// TIA Portal V16 export
// export: Created 2023-01-31T04:00:58.1302964Z, ExportSetting WithDefaults, WithReadOnly, DisplayName Totally Integrated Automation Portal, DisplayVersion V16 Update 1, DisplayName TIA Portal Version Control Interface, DisplayVersion V16, DisplayName TIA Portal Openness, DisplayVersion V16 Update 1, DisplayName SINAMICS Startdrive Advanced, DisplayVersion V16, DisplayName SINAMICS Startdrive G130, G150, S120, S150, SINAMICS MV, S210, DisplayVersion V16, DisplayName SINAMICS Startdrive G110M, G120, G120C, G120D, G120P, DisplayVersion V16, DisplayName STEP 7 Professional, DisplayVersion V16 Update 1, DisplayName STEP 7 Safety, DisplayVersion V16, DisplayName WinCC Advanced, DisplayVersion V16 Update 1
FUNCTION "022SAE001_Call" : Void   // FC80, LAD
TITLE = 022SAE001 Deposit 1 / 010ABS001 Ablage 1
{ S7_Optimized_Access := 'FALSE' }
VERSION : 0.1
// stored: AutoNumber true, CodeModifiedDate 2021-01-26T01:38:20.3874578Z, CompileDate 2021-02-05T02:55:14.1436684Z, CreationDate 2019-06-27T08:21:26.7500417Z, HandleErrorsWithinBlock false, InterfaceModifiedDate 2017-10-27T11:23:23.7919428Z, IsConsistent true, IsIECCheckEnabled false, IsKnowHowProtected false, IsWriteProtected false, LibraryConformanceStatus Error: The block contains calls of single instances. Warning: The object contains access to global data blocks. Warning: The block contains direct access to inputs, outputs, bit memories, indirect access to the registry or indirect access to external memory areas that are unknown at the time of compilation., ModifiedDate 2021-01-26T01:38:20.3874578Z, ParameterModified 2017-10-27T11:23:23.7469402Z, PLCSimAdvancedSupport true, SetENOAutomatically false, StructureModified 2017-10-27T11:23:23.7919428Z, UDAEnableTagReadback false
   VAR_TEMP   // added for the SCL form of the ladder/FBD networks
      _w1 : Bool;
      _s5time1 : S5Time;
   END_VAR
BEGIN

REGION Network 1: 022SAE001-BZ1.1 part control
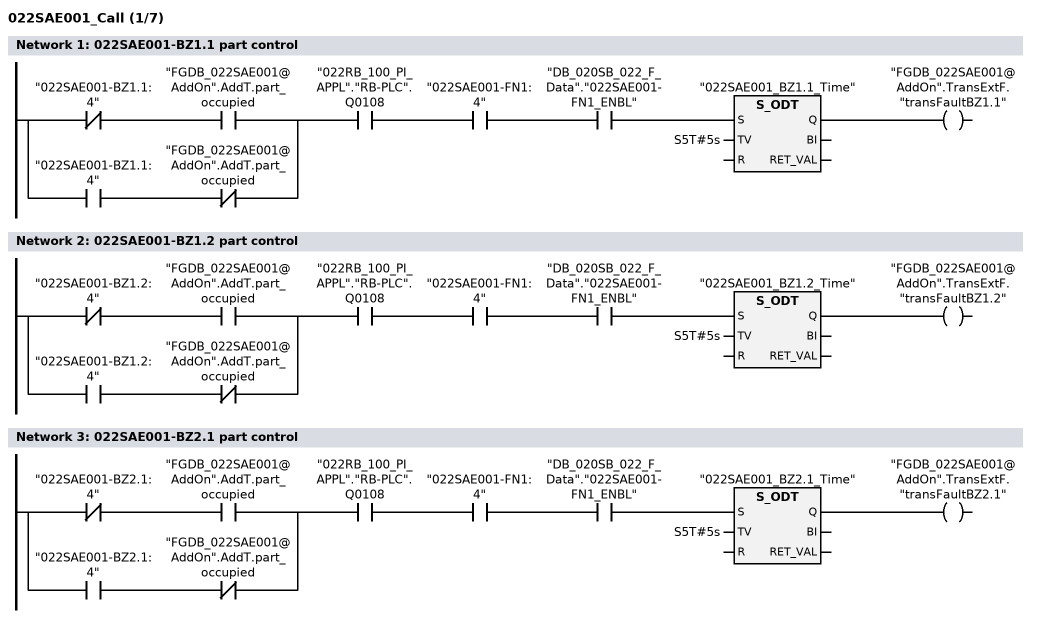
   RUNG wire#powerrail
      I_Contact( "022SAE001-BZ1.1:4" )
      Contact( "FGDB_022SAE001@AddOn".AddT.part_occupied )
      wire#w1
      Contact( "022RB_100_PI_APPL"."RB-PLC".Q0108 )
      Contact( "022SAE001-FN1:4" )
      Contact( "DB_020SB_022_F_Data"."022SAE001-FN1_ENBL" )
      S_ODT(T_NO := "022SAE001_BZ1.1_Time", TV := S5T#5s, R :=, BI =>, RET_VAL =>)
      Coil( "FGDB_022SAE001@AddOn".TransExtF."transFaultBZ1.1" )
   END_RUNG
   RUNG wire#powerrail
      Contact( "022SAE001-BZ1.1:4" )
      I_Contact( "FGDB_022SAE001@AddOn".AddT.part_occupied )
   END_RUNG wire#w1
   // the same network as SCL:
   #_s5time1 := S_ODT(T_NO := "022SAE001_BZ1.1_Time",
                      S := ((NOT "022SAE001-BZ1.1:4" AND "FGDB_022SAE001@AddOn".AddT.part_occupied) OR ("022SAE001-BZ1.1:4" AND NOT "FGDB_022SAE001@AddOn".AddT.part_occupied)) AND "022RB_100_PI_APPL"."RB-PLC".Q0108 AND "022SAE001-FN1:4" AND "DB_020SB_022_F_Data"."022SAE001-FN1_ENBL",
                      TV := S5T#5s,
                      Q => #_w1);
   "FGDB_022SAE001@AddOn".TransExtF."transFaultBZ1.1" := #_w1;
END_REGION

REGION Network 2: 022SAE001-BZ1.2 part control
   RUNG wire#powerrail
      I_Contact( "022SAE001-BZ1.2:4" )
      Contact( "FGDB_022SAE001@AddOn".AddT.part_occupied )
      wire#w1
      Contact( "022RB_100_PI_APPL"."RB-PLC".Q0108 )
      Contact( "022SAE001-FN1:4" )
      Contact( "DB_020SB_022_F_Data"."022SAE001-FN1_ENBL" )
      S_ODT(T_NO := "022SAE001_BZ1.2_Time", TV := S5T#5s, R :=, BI =>, RET_VAL =>)
      Coil( "FGDB_022SAE001@AddOn".TransExtF."transFaultBZ1.2" )
   END_RUNG
   RUNG wire#powerrail
      Contact( "022SAE001-BZ1.2:4" )
      I_Contact( "FGDB_022SAE001@AddOn".AddT.part_occupied )
   END_RUNG wire#w1
   // the same network as SCL:
   #_s5time1 := S_ODT(T_NO := "022SAE001_BZ1.2_Time",
                      S := ((NOT "022SAE001-BZ1.2:4" AND "FGDB_022SAE001@AddOn".AddT.part_occupied) OR ("022SAE001-BZ1.2:4" AND NOT "FGDB_022SAE001@AddOn".AddT.part_occupied)) AND "022RB_100_PI_APPL"."RB-PLC".Q0108 AND "022SAE001-FN1:4" AND "DB_020SB_022_F_Data"."022SAE001-FN1_ENBL",
                      TV := S5T#5s,
                      Q => #_w1);
   "FGDB_022SAE001@AddOn".TransExtF."transFaultBZ1.2" := #_w1;
END_REGION

REGION Network 3: 022SAE001-BZ2.1 part control
   RUNG wire#powerrail
      I_Contact( "022SAE001-BZ2.1:4" )
      Contact( "FGDB_022SAE001@AddOn".AddT.part_occupied )
      wire#w1
      Contact( "022RB_100_PI_APPL"."RB-PLC".Q0108 )
      Contact( "022SAE001-FN1:4" )
      Contact( "DB_020SB_022_F_Data"."022SAE001-FN1_ENBL" )
      S_ODT(T_NO := "022SAE001_BZ2.1_Time", TV := S5T#5s, R :=, BI =>, RET_VAL =>)
      Coil( "FGDB_022SAE001@AddOn".TransExtF."transFaultBZ2.1" )
   END_RUNG
   RUNG wire#powerrail
      Contact( "022SAE001-BZ2.1:4" )
      I_Contact( "FGDB_022SAE001@AddOn".AddT.part_occupied )
   END_RUNG wire#w1
   // the same network as SCL:
   #_s5time1 := S_ODT(T_NO := "022SAE001_BZ2.1_Time",
                      S := ((NOT "022SAE001-BZ2.1:4" AND "FGDB_022SAE001@AddOn".AddT.part_occupied) OR ("022SAE001-BZ2.1:4" AND NOT "FGDB_022SAE001@AddOn".AddT.part_occupied)) AND "022RB_100_PI_APPL"."RB-PLC".Q0108 AND "022SAE001-FN1:4" AND "DB_020SB_022_F_Data"."022SAE001-FN1_ENBL",
                      TV := S5T#5s,
                      Q => #_w1);
   "FGDB_022SAE001@AddOn".TransExtF."transFaultBZ2.1" := #_w1;
END_REGION

REGION Network 4: Enter additional malfunctions 022SAE001
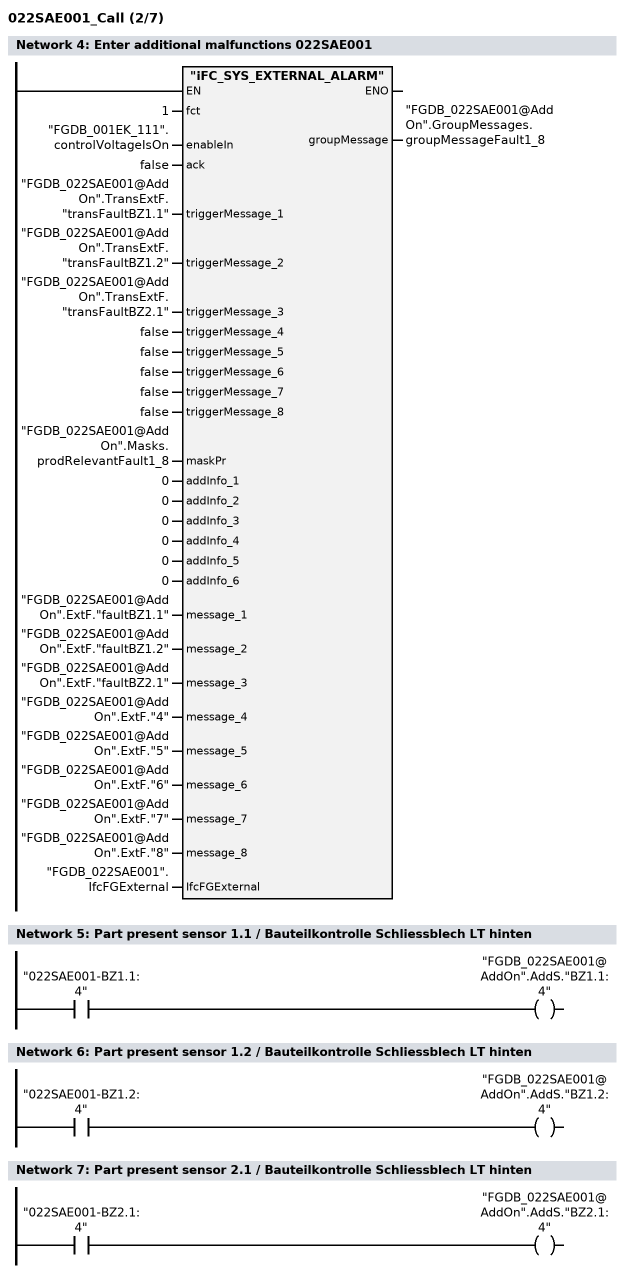
   RUNG wire#powerrail
      "iFC_SYS_EXTERNAL_ALARM"(fct := 1, enableIn := "FGDB_001EK_111".controlVoltageIsOn, ack := false, triggerMessage_1 := "FGDB_022SAE001@AddOn".TransExtF."transFaultBZ1.1", triggerMessage_2 := "FGDB_022SAE001@AddOn".TransExtF."transFaultBZ1.2", triggerMessage_3 := "FGDB_022SAE001@AddOn".TransExtF."transFaultBZ2.1", triggerMessage_4 := false, triggerMessage_5 := false, triggerMessage_6 := false, triggerMessage_7 := false, triggerMessage_8 := false, maskPr := "FGDB_022SAE001@AddOn".Masks.prodRelevantFault1_8, addInfo_1 := 0, addInfo_2 := 0, addInfo_3 := 0, addInfo_4 := 0, addInfo_5 := 0, addInfo_6 := 0, message_1 := "FGDB_022SAE001@AddOn".ExtF."faultBZ1.1", message_2 := "FGDB_022SAE001@AddOn".ExtF."faultBZ1.2", message_3 := "FGDB_022SAE001@AddOn".ExtF."faultBZ2.1", message_4 := "FGDB_022SAE001@AddOn".ExtF."4", message_5 := "FGDB_022SAE001@AddOn".ExtF."5", message_6 := "FGDB_022SAE001@AddOn".ExtF."6", message_7 := "FGDB_022SAE001@AddOn".ExtF."7", message_8 := "FGDB_022SAE001@AddOn".ExtF."8", IfcFGExternal := "FGDB_022SAE001".IfcFGExternal, groupMessage => "FGDB_022SAE001@AddOn".GroupMessages.groupMessageFault1_8)
   END_RUNG
   // the same network as SCL:
   "iFC_SYS_EXTERNAL_ALARM"(fct := 1,
                           enableIn := "FGDB_001EK_111".controlVoltageIsOn,
                           ack := false,
                           triggerMessage_1 := "FGDB_022SAE001@AddOn".TransExtF."transFaultBZ1.1",
                           triggerMessage_2 := "FGDB_022SAE001@AddOn".TransExtF."transFaultBZ1.2",
                           triggerMessage_3 := "FGDB_022SAE001@AddOn".TransExtF."transFaultBZ2.1",
                           triggerMessage_4 := false,
                           triggerMessage_5 := false,
                           triggerMessage_6 := false,
                           triggerMessage_7 := false,
                           triggerMessage_8 := false,
                           maskPr := "FGDB_022SAE001@AddOn".Masks.prodRelevantFault1_8,
                           addInfo_1 := 0,
                           addInfo_2 := 0,
                           addInfo_3 := 0,
                           addInfo_4 := 0,
                           addInfo_5 := 0,
                           addInfo_6 := 0,
                           message_1 := "FGDB_022SAE001@AddOn".ExtF."faultBZ1.1",
                           message_2 := "FGDB_022SAE001@AddOn".ExtF."faultBZ1.2",
                           message_3 := "FGDB_022SAE001@AddOn".ExtF."faultBZ2.1",
                           message_4 := "FGDB_022SAE001@AddOn".ExtF."4",
                           message_5 := "FGDB_022SAE001@AddOn".ExtF."5",
                           message_6 := "FGDB_022SAE001@AddOn".ExtF."6",
                           message_7 := "FGDB_022SAE001@AddOn".ExtF."7",
                           message_8 := "FGDB_022SAE001@AddOn".ExtF."8",
                           IfcFGExternal := "FGDB_022SAE001".IfcFGExternal,
                           groupMessage => "FGDB_022SAE001@AddOn".GroupMessages.groupMessageFault1_8);
END_REGION

REGION Network 5: Part present sensor 1.1 / Bauteilkontrolle Schliessblech LT hinten
   RUNG wire#powerrail
      Contact( "022SAE001-BZ1.1:4" )
      Coil( "FGDB_022SAE001@AddOn".AddS."BZ1.1:4" )
   END_RUNG
   // the same network as SCL:
   "FGDB_022SAE001@AddOn".AddS."BZ1.1:4" := "022SAE001-BZ1.1:4";
END_REGION

REGION Network 6: Part present sensor 1.2 / Bauteilkontrolle Schliessblech LT hinten
   RUNG wire#powerrail
      Contact( "022SAE001-BZ1.2:4" )
      Coil( "FGDB_022SAE001@AddOn".AddS."BZ1.2:4" )
   END_RUNG
   // the same network as SCL:
   "FGDB_022SAE001@AddOn".AddS."BZ1.2:4" := "022SAE001-BZ1.2:4";
END_REGION

REGION Network 7: Part present sensor 2.1 / Bauteilkontrolle Schliessblech LT hinten
   RUNG wire#powerrail
      Contact( "022SAE001-BZ2.1:4" )
      Coil( "FGDB_022SAE001@AddOn".AddS."BZ2.1:4" )
   END_RUNG
   // the same network as SCL:
   "FGDB_022SAE001@AddOn".AddS."BZ2.1:4" := "022SAE001-BZ2.1:4";
END_REGION

REGION Network 8: 022SAE001 Part1 occupied / Teil belegt Federbeintopf
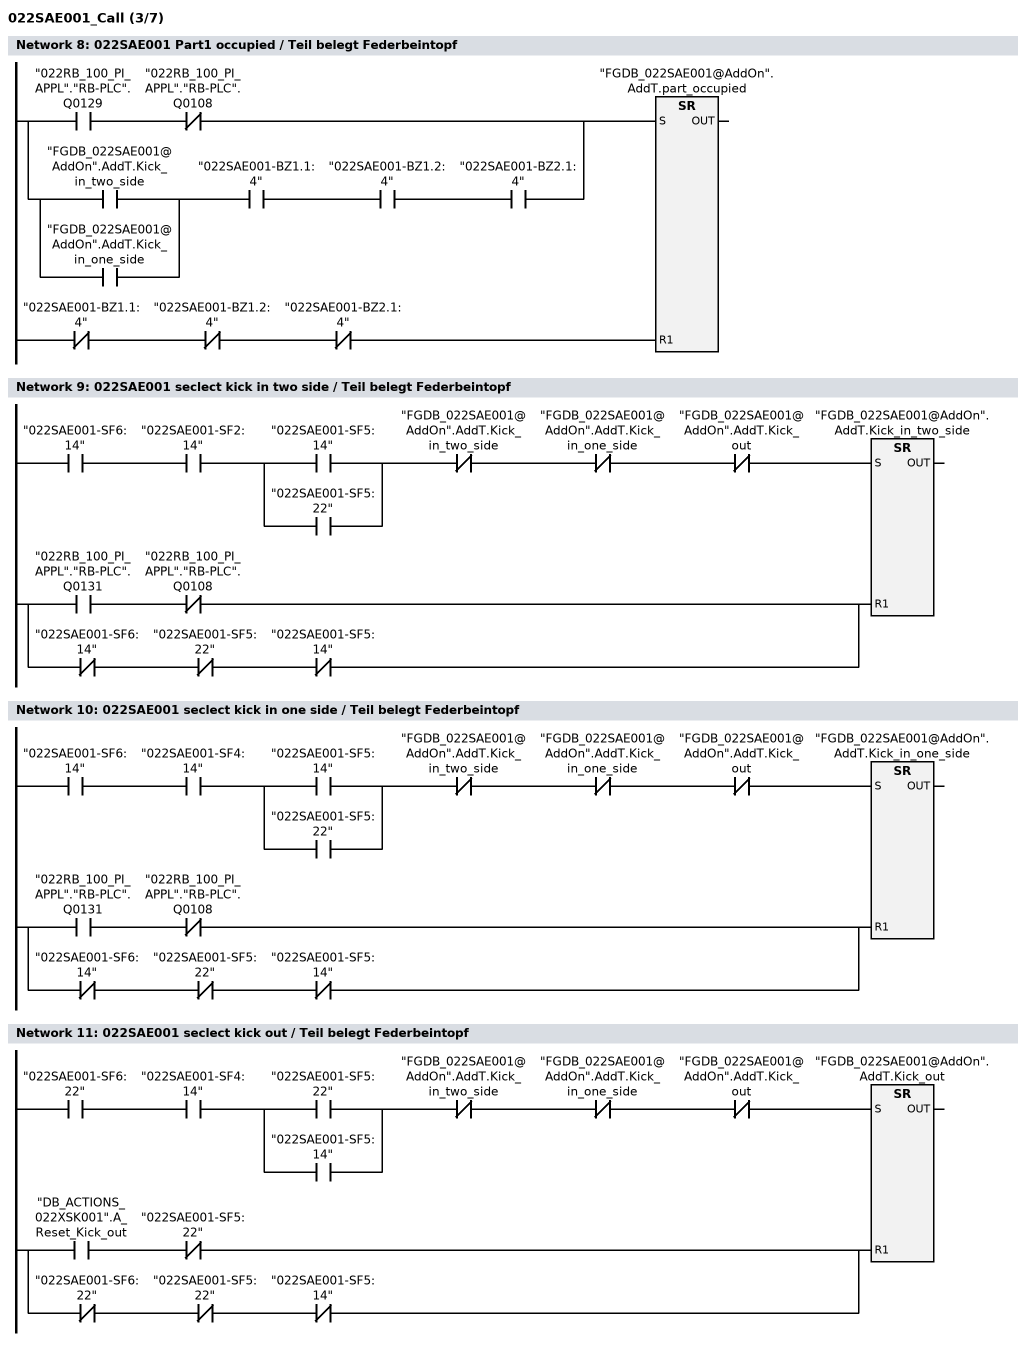
   RUNG wire#powerrail
      Contact( "022RB_100_PI_APPL"."RB-PLC".Q0129 )
      I_Contact( "022RB_100_PI_APPL"."RB-PLC".Q0108 )
      wire#w1
      S_SR(operand := "FGDB_022SAE001@AddOn".AddT.part_occupied, r1 := wire#w3)
   END_RUNG
   RUNG wire#powerrail
      Contact( "FGDB_022SAE001@AddOn".AddT.Kick_in_two_side )
      wire#w2
      Contact( "022SAE001-BZ1.1:4" )
      Contact( "022SAE001-BZ1.2:4" )
      Contact( "022SAE001-BZ2.1:4" )
   END_RUNG wire#w1
   RUNG wire#powerrail
      Contact( "FGDB_022SAE001@AddOn".AddT.Kick_in_one_side )
   END_RUNG wire#w2
   RUNG wire#powerrail
      I_Contact( "022SAE001-BZ1.1:4" )
      I_Contact( "022SAE001-BZ1.2:4" )
      I_Contact( "022SAE001-BZ2.1:4" )
   END_RUNG wire#w3
   // the same network as SCL:
   IF ("022RB_100_PI_APPL"."RB-PLC".Q0129 AND NOT "022RB_100_PI_APPL"."RB-PLC".Q0108) OR (("FGDB_022SAE001@AddOn".AddT.Kick_in_two_side OR "FGDB_022SAE001@AddOn".AddT.Kick_in_one_side) AND "022SAE001-BZ1.1:4" AND "022SAE001-BZ1.2:4" AND "022SAE001-BZ2.1:4") THEN
       "FGDB_022SAE001@AddOn".AddT.part_occupied := TRUE;   // SR flip-flop
   END_IF;
   IF NOT "022SAE001-BZ1.1:4" AND NOT "022SAE001-BZ1.2:4" AND NOT "022SAE001-BZ2.1:4" THEN
       "FGDB_022SAE001@AddOn".AddT.part_occupied := FALSE;
   END_IF;
END_REGION

REGION Network 9: 022SAE001 seclect kick in two side / Teil belegt Federbeintopf
   RUNG wire#powerrail
      Contact( "022SAE001-SF6:14" )
      Contact( "022SAE001-SF2:14" )
      wire#w1
      Contact( "022SAE001-SF5:14" )
      wire#w2
      I_Contact( "FGDB_022SAE001@AddOn".AddT.Kick_in_two_side )
      I_Contact( "FGDB_022SAE001@AddOn".AddT.Kick_in_one_side )
      I_Contact( "FGDB_022SAE001@AddOn".AddT.Kick_out )
      S_SR(operand := "FGDB_022SAE001@AddOn".AddT.Kick_in_two_side, r1 := wire#w3)
   END_RUNG
   RUNG wire#w1
      Contact( "022SAE001-SF5:22" )
   END_RUNG wire#w2
   RUNG wire#powerrail
      Contact( "022RB_100_PI_APPL"."RB-PLC".Q0131 )
      I_Contact( "022RB_100_PI_APPL"."RB-PLC".Q0108 )
   END_RUNG wire#w3
   RUNG wire#powerrail
      I_Contact( "022SAE001-SF6:14" )
      I_Contact( "022SAE001-SF5:22" )
      I_Contact( "022SAE001-SF5:14" )
   END_RUNG wire#w3
   // the same network as SCL:
   IF "022SAE001-SF6:14" AND "022SAE001-SF2:14" AND ("022SAE001-SF5:14" OR "022SAE001-SF5:22") AND NOT "FGDB_022SAE001@AddOn".AddT.Kick_in_two_side AND NOT "FGDB_022SAE001@AddOn".AddT.Kick_in_one_side AND NOT "FGDB_022SAE001@AddOn".AddT.Kick_out THEN
       "FGDB_022SAE001@AddOn".AddT.Kick_in_two_side := TRUE;   // SR flip-flop
   END_IF;
   IF ("022RB_100_PI_APPL"."RB-PLC".Q0131 AND NOT "022RB_100_PI_APPL"."RB-PLC".Q0108) OR (NOT "022SAE001-SF6:14" AND NOT "022SAE001-SF5:22" AND NOT "022SAE001-SF5:14") THEN
       "FGDB_022SAE001@AddOn".AddT.Kick_in_two_side := FALSE;
   END_IF;
END_REGION

REGION Network 10: 022SAE001 seclect kick in one side / Teil belegt Federbeintopf
   RUNG wire#powerrail
      Contact( "022SAE001-SF6:14" )
      Contact( "022SAE001-SF4:14" )
      wire#w1
      Contact( "022SAE001-SF5:14" )
      wire#w2
      I_Contact( "FGDB_022SAE001@AddOn".AddT.Kick_in_two_side )
      I_Contact( "FGDB_022SAE001@AddOn".AddT.Kick_in_one_side )
      I_Contact( "FGDB_022SAE001@AddOn".AddT.Kick_out )
      S_SR(operand := "FGDB_022SAE001@AddOn".AddT.Kick_in_one_side, r1 := wire#w3)
   END_RUNG
   RUNG wire#w1
      Contact( "022SAE001-SF5:22" )
   END_RUNG wire#w2
   RUNG wire#powerrail
      Contact( "022RB_100_PI_APPL"."RB-PLC".Q0131 )
      I_Contact( "022RB_100_PI_APPL"."RB-PLC".Q0108 )
   END_RUNG wire#w3
   RUNG wire#powerrail
      I_Contact( "022SAE001-SF6:14" )
      I_Contact( "022SAE001-SF5:22" )
      I_Contact( "022SAE001-SF5:14" )
   END_RUNG wire#w3
   // the same network as SCL:
   IF "022SAE001-SF6:14" AND "022SAE001-SF4:14" AND ("022SAE001-SF5:14" OR "022SAE001-SF5:22") AND NOT "FGDB_022SAE001@AddOn".AddT.Kick_in_two_side AND NOT "FGDB_022SAE001@AddOn".AddT.Kick_in_one_side AND NOT "FGDB_022SAE001@AddOn".AddT.Kick_out THEN
       "FGDB_022SAE001@AddOn".AddT.Kick_in_one_side := TRUE;   // SR flip-flop
   END_IF;
   IF ("022RB_100_PI_APPL"."RB-PLC".Q0131 AND NOT "022RB_100_PI_APPL"."RB-PLC".Q0108) OR (NOT "022SAE001-SF6:14" AND NOT "022SAE001-SF5:22" AND NOT "022SAE001-SF5:14") THEN
       "FGDB_022SAE001@AddOn".AddT.Kick_in_one_side := FALSE;
   END_IF;
END_REGION

REGION Network 11: 022SAE001 seclect kick out / Teil belegt Federbeintopf
   RUNG wire#powerrail
      Contact( "022SAE001-SF6:22" )
      Contact( "022SAE001-SF4:14" )
      wire#w1
      Contact( "022SAE001-SF5:22" )
      wire#w2
      I_Contact( "FGDB_022SAE001@AddOn".AddT.Kick_in_two_side )
      I_Contact( "FGDB_022SAE001@AddOn".AddT.Kick_in_one_side )
      I_Contact( "FGDB_022SAE001@AddOn".AddT.Kick_out )
      S_SR(operand := "FGDB_022SAE001@AddOn".AddT.Kick_out, r1 := wire#w3)
   END_RUNG
   RUNG wire#w1
      Contact( "022SAE001-SF5:14" )
   END_RUNG wire#w2
   RUNG wire#powerrail
      Contact( "DB_ACTIONS_022XSK001".A_Reset_Kick_out )
      I_Contact( "022SAE001-SF5:22" )
   END_RUNG wire#w3
   RUNG wire#powerrail
      I_Contact( "022SAE001-SF6:22" )
      I_Contact( "022SAE001-SF5:22" )
      I_Contact( "022SAE001-SF5:14" )
   END_RUNG wire#w3
   // the same network as SCL:
   IF "022SAE001-SF6:22" AND "022SAE001-SF4:14" AND ("022SAE001-SF5:22" OR "022SAE001-SF5:14") AND NOT "FGDB_022SAE001@AddOn".AddT.Kick_in_two_side AND NOT "FGDB_022SAE001@AddOn".AddT.Kick_in_one_side AND NOT "FGDB_022SAE001@AddOn".AddT.Kick_out THEN
       "FGDB_022SAE001@AddOn".AddT.Kick_out := TRUE;   // SR flip-flop
   END_IF;
   IF ("DB_ACTIONS_022XSK001".A_Reset_Kick_out AND NOT "022SAE001-SF5:22") OR (NOT "022SAE001-SF6:22" AND NOT "022SAE001-SF5:22" AND NOT "022SAE001-SF5:14") THEN
       "FGDB_022SAE001@AddOn".AddT.Kick_out := FALSE;
   END_IF;
END_REGION

REGION Network 12: 022SAE001 initial position station empty
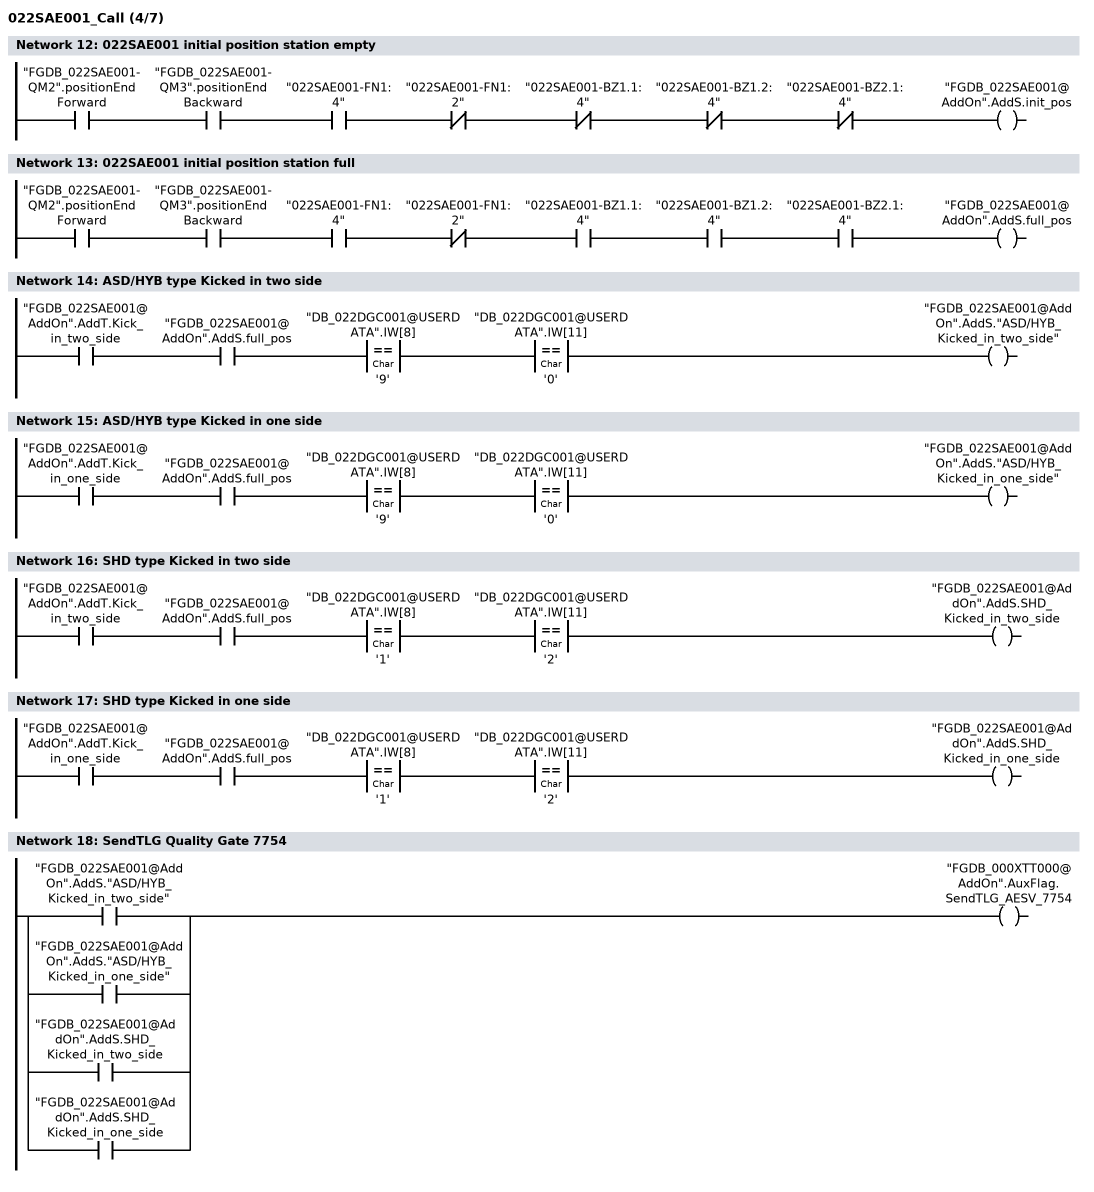
   RUNG wire#powerrail
      Contact( "FGDB_022SAE001-QM2".positionEndForward )
      Contact( "FGDB_022SAE001-QM3".positionEndBackward )
      Contact( "022SAE001-FN1:4" )
      I_Contact( "022SAE001-FN1:2" )
      I_Contact( "022SAE001-BZ1.1:4" )
      I_Contact( "022SAE001-BZ1.2:4" )
      I_Contact( "022SAE001-BZ2.1:4" )
      Coil( "FGDB_022SAE001@AddOn".AddS.init_pos )
   END_RUNG
   // the same network as SCL:
   "FGDB_022SAE001@AddOn".AddS.init_pos := "FGDB_022SAE001-QM2".positionEndForward AND "FGDB_022SAE001-QM3".positionEndBackward AND "022SAE001-FN1:4" AND NOT "022SAE001-FN1:2" AND NOT "022SAE001-BZ1.1:4" AND NOT "022SAE001-BZ1.2:4" AND NOT "022SAE001-BZ2.1:4";
END_REGION

REGION Network 13: 022SAE001 initial position station full
   RUNG wire#powerrail
      Contact( "FGDB_022SAE001-QM2".positionEndForward )
      Contact( "FGDB_022SAE001-QM3".positionEndBackward )
      Contact( "022SAE001-FN1:4" )
      I_Contact( "022SAE001-FN1:2" )
      Contact( "022SAE001-BZ1.1:4" )
      Contact( "022SAE001-BZ1.2:4" )
      Contact( "022SAE001-BZ2.1:4" )
      Coil( "FGDB_022SAE001@AddOn".AddS.full_pos )
   END_RUNG
   // the same network as SCL:
   "FGDB_022SAE001@AddOn".AddS.full_pos := "FGDB_022SAE001-QM2".positionEndForward AND "FGDB_022SAE001-QM3".positionEndBackward AND "022SAE001-FN1:4" AND NOT "022SAE001-FN1:2" AND "022SAE001-BZ1.1:4" AND "022SAE001-BZ1.2:4" AND "022SAE001-BZ2.1:4";
END_REGION

REGION Network 14: ASD/HYB type Kicked in two side
   RUNG wire#powerrail
      Contact( "FGDB_022SAE001@AddOn".AddT.Kick_in_two_side )
      Contact( "FGDB_022SAE001@AddOn".AddS.full_pos )
      { S7_Templates := "SrcType := Char" } EQ_Contact(in1 := "DB_022DGC001@USERDATA".IW[8], in2 := '9')
      { S7_Templates := "SrcType := Char" } EQ_Contact(in1 := "DB_022DGC001@USERDATA".IW[11], in2 := '0')
      Coil( "FGDB_022SAE001@AddOn".AddS."ASD/HYB_Kicked_in_two_side" )
   END_RUNG
   // the same network as SCL:
   "FGDB_022SAE001@AddOn".AddS."ASD/HYB_Kicked_in_two_side" := "FGDB_022SAE001@AddOn".AddT.Kick_in_two_side AND "FGDB_022SAE001@AddOn".AddS.full_pos AND ("DB_022DGC001@USERDATA".IW[8] = '9') AND ("DB_022DGC001@USERDATA".IW[11] = '0');
END_REGION

REGION Network 15: ASD/HYB type Kicked in one side
   RUNG wire#powerrail
      Contact( "FGDB_022SAE001@AddOn".AddT.Kick_in_one_side )
      Contact( "FGDB_022SAE001@AddOn".AddS.full_pos )
      { S7_Templates := "SrcType := Char" } EQ_Contact(in1 := "DB_022DGC001@USERDATA".IW[8], in2 := '9')
      { S7_Templates := "SrcType := Char" } EQ_Contact(in1 := "DB_022DGC001@USERDATA".IW[11], in2 := '0')
      Coil( "FGDB_022SAE001@AddOn".AddS."ASD/HYB_Kicked_in_one_side" )
   END_RUNG
   // the same network as SCL:
   "FGDB_022SAE001@AddOn".AddS."ASD/HYB_Kicked_in_one_side" := "FGDB_022SAE001@AddOn".AddT.Kick_in_one_side AND "FGDB_022SAE001@AddOn".AddS.full_pos AND ("DB_022DGC001@USERDATA".IW[8] = '9') AND ("DB_022DGC001@USERDATA".IW[11] = '0');
END_REGION

REGION Network 16: SHD type Kicked in two side
   RUNG wire#powerrail
      Contact( "FGDB_022SAE001@AddOn".AddT.Kick_in_two_side )
      Contact( "FGDB_022SAE001@AddOn".AddS.full_pos )
      { S7_Templates := "SrcType := Char" } EQ_Contact(in1 := "DB_022DGC001@USERDATA".IW[8], in2 := '1')
      { S7_Templates := "SrcType := Char" } EQ_Contact(in1 := "DB_022DGC001@USERDATA".IW[11], in2 := '2')
      Coil( "FGDB_022SAE001@AddOn".AddS.SHD_Kicked_in_two_side )
   END_RUNG
   // the same network as SCL:
   "FGDB_022SAE001@AddOn".AddS.SHD_Kicked_in_two_side := "FGDB_022SAE001@AddOn".AddT.Kick_in_two_side AND "FGDB_022SAE001@AddOn".AddS.full_pos AND ("DB_022DGC001@USERDATA".IW[8] = '1') AND ("DB_022DGC001@USERDATA".IW[11] = '2');
END_REGION

REGION Network 17: SHD type Kicked in one side
   RUNG wire#powerrail
      Contact( "FGDB_022SAE001@AddOn".AddT.Kick_in_one_side )
      Contact( "FGDB_022SAE001@AddOn".AddS.full_pos )
      { S7_Templates := "SrcType := Char" } EQ_Contact(in1 := "DB_022DGC001@USERDATA".IW[8], in2 := '1')
      { S7_Templates := "SrcType := Char" } EQ_Contact(in1 := "DB_022DGC001@USERDATA".IW[11], in2 := '2')
      Coil( "FGDB_022SAE001@AddOn".AddS.SHD_Kicked_in_one_side )
   END_RUNG
   // the same network as SCL:
   "FGDB_022SAE001@AddOn".AddS.SHD_Kicked_in_one_side := "FGDB_022SAE001@AddOn".AddT.Kick_in_one_side AND "FGDB_022SAE001@AddOn".AddS.full_pos AND ("DB_022DGC001@USERDATA".IW[8] = '1') AND ("DB_022DGC001@USERDATA".IW[11] = '2');
END_REGION

REGION Network 18: SendTLG Quality Gate 7754
   RUNG wire#powerrail
      Contact( "FGDB_022SAE001@AddOn".AddS."ASD/HYB_Kicked_in_two_side" )
      wire#w1
      Coil( "FGDB_000XTT000@AddOn".AuxFlag.SendTLG_AESV_7754 )
   END_RUNG
   RUNG wire#powerrail
      Contact( "FGDB_022SAE001@AddOn".AddS."ASD/HYB_Kicked_in_one_side" )
   END_RUNG wire#w1
   RUNG wire#powerrail
      Contact( "FGDB_022SAE001@AddOn".AddS.SHD_Kicked_in_two_side )
   END_RUNG wire#w1
   RUNG wire#powerrail
      Contact( "FGDB_022SAE001@AddOn".AddS.SHD_Kicked_in_one_side )
   END_RUNG wire#w1
   // the same network as SCL:
   "FGDB_000XTT000@AddOn".AuxFlag.SendTLG_AESV_7754 := "FGDB_022SAE001@AddOn".AddS."ASD/HYB_Kicked_in_two_side" OR "FGDB_022SAE001@AddOn".AddS."ASD/HYB_Kicked_in_one_side" OR "FGDB_022SAE001@AddOn".AddS.SHD_Kicked_in_two_side OR "FGDB_022SAE001@AddOn".AddS.SHD_Kicked_in_one_side;
END_REGION

REGION Network 19: Q-gate quality feedback ok
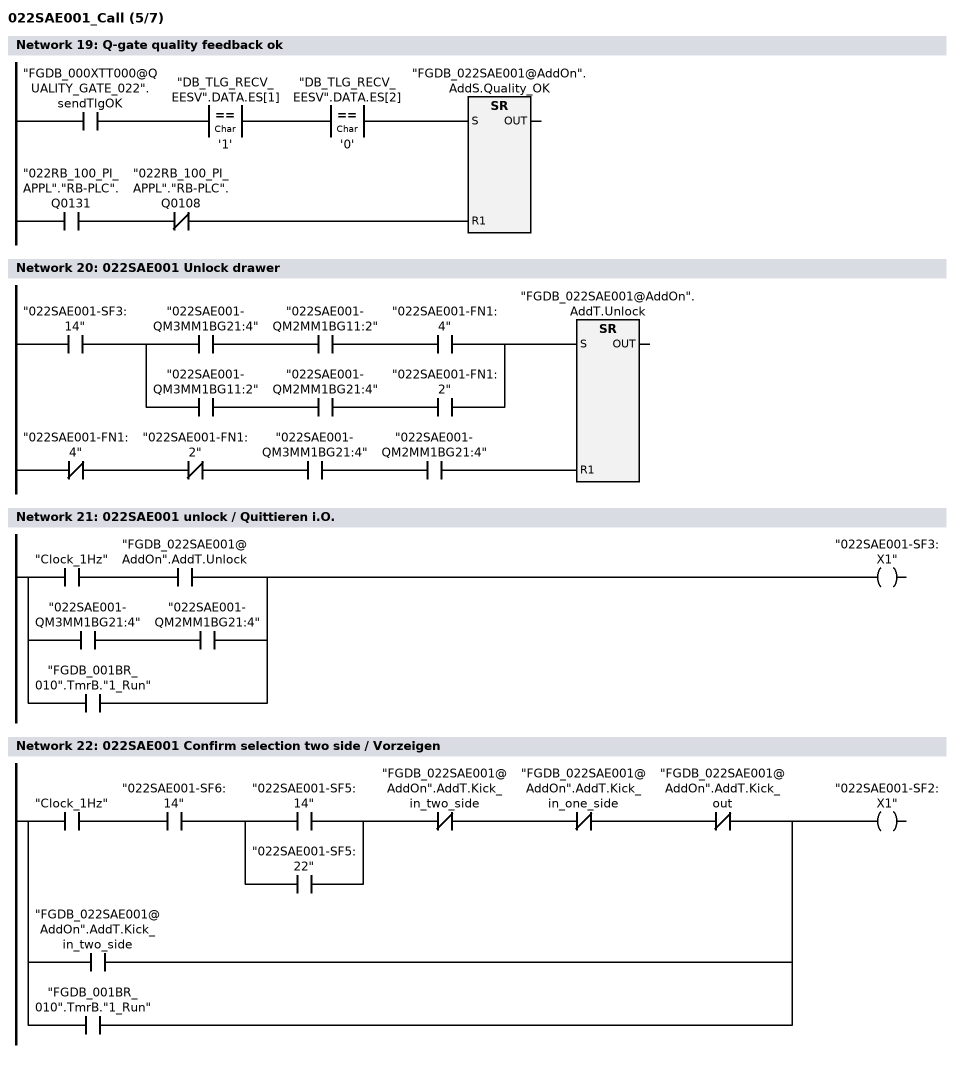
   RUNG wire#powerrail
      Contact( "FGDB_000XTT000@QUALITY_GATE_022".sendTlgOK )
      { S7_Templates := "SrcType := Char" } EQ_Contact(in1 := "DB_TLG_RECV_EESV".DATA.ES[1], in2 := '1')
      { S7_Templates := "SrcType := Char" } EQ_Contact(in1 := "DB_TLG_RECV_EESV".DATA.ES[2], in2 := '0')
      S_SR(operand := "FGDB_022SAE001@AddOn".AddS.Quality_OK, r1 := wire#w1)
   END_RUNG
   RUNG wire#powerrail
      Contact( "022RB_100_PI_APPL"."RB-PLC".Q0131 )
      I_Contact( "022RB_100_PI_APPL"."RB-PLC".Q0108 )
   END_RUNG wire#w1
   // the same network as SCL:
   IF "FGDB_000XTT000@QUALITY_GATE_022".sendTlgOK AND ("DB_TLG_RECV_EESV".DATA.ES[1] = '1') AND ("DB_TLG_RECV_EESV".DATA.ES[2] = '0') THEN
       "FGDB_022SAE001@AddOn".AddS.Quality_OK := TRUE;   // SR flip-flop
   END_IF;
   IF "022RB_100_PI_APPL"."RB-PLC".Q0131 AND NOT "022RB_100_PI_APPL"."RB-PLC".Q0108 THEN
       "FGDB_022SAE001@AddOn".AddS.Quality_OK := FALSE;
   END_IF;
END_REGION

REGION Network 20: 022SAE001 Unlock drawer
   RUNG wire#powerrail
      Contact( "022SAE001-SF3:14" )
      wire#w1
      Contact( "022SAE001-QM3MM1BG21:4" )
      Contact( "022SAE001-QM2MM1BG11:2" )
      Contact( "022SAE001-FN1:4" )
      wire#w2
      S_SR(operand := "FGDB_022SAE001@AddOn".AddT.Unlock, r1 := wire#w3)
   END_RUNG
   RUNG wire#w1
      Contact( "022SAE001-QM3MM1BG11:2" )
      Contact( "022SAE001-QM2MM1BG21:4" )
      Contact( "022SAE001-FN1:2" )
   END_RUNG wire#w2
   RUNG wire#powerrail
      I_Contact( "022SAE001-FN1:4" )
      I_Contact( "022SAE001-FN1:2" )
      Contact( "022SAE001-QM3MM1BG21:4" )
      Contact( "022SAE001-QM2MM1BG21:4" )
   END_RUNG wire#w3
   // the same network as SCL:
   IF "022SAE001-SF3:14" AND (("022SAE001-QM3MM1BG21:4" AND "022SAE001-QM2MM1BG11:2" AND "022SAE001-FN1:4") OR ("022SAE001-QM3MM1BG11:2" AND "022SAE001-QM2MM1BG21:4" AND "022SAE001-FN1:2")) THEN
       "FGDB_022SAE001@AddOn".AddT.Unlock := TRUE;   // SR flip-flop
   END_IF;
   IF NOT "022SAE001-FN1:4" AND NOT "022SAE001-FN1:2" AND "022SAE001-QM3MM1BG21:4" AND "022SAE001-QM2MM1BG21:4" THEN
       "FGDB_022SAE001@AddOn".AddT.Unlock := FALSE;
   END_IF;
END_REGION

REGION Network 21: 022SAE001 unlock / Quittieren i.O.
   RUNG wire#powerrail
      Contact( "Clock_1Hz" )
      Contact( "FGDB_022SAE001@AddOn".AddT.Unlock )
      wire#w1
      Coil( "022SAE001-SF3:X1" )
   END_RUNG
   RUNG wire#powerrail
      Contact( "022SAE001-QM3MM1BG21:4" )
      Contact( "022SAE001-QM2MM1BG21:4" )
   END_RUNG wire#w1
   RUNG wire#powerrail
      Contact( "FGDB_001BR_010".TmrB."1_Run" )
   END_RUNG wire#w1
   // the same network as SCL:
   "022SAE001-SF3:X1" := ("Clock_1Hz" AND "FGDB_022SAE001@AddOn".AddT.Unlock) OR ("022SAE001-QM3MM1BG21:4" AND "022SAE001-QM2MM1BG21:4") OR "FGDB_001BR_010".TmrB."1_Run";
END_REGION

REGION Network 22: 022SAE001 Confirm selection two side / Vorzeigen
   RUNG wire#powerrail
      Contact( "Clock_1Hz" )
      Contact( "022SAE001-SF6:14" )
      wire#w1
      Contact( "022SAE001-SF5:14" )
      wire#w2
      I_Contact( "FGDB_022SAE001@AddOn".AddT.Kick_in_two_side )
      I_Contact( "FGDB_022SAE001@AddOn".AddT.Kick_in_one_side )
      I_Contact( "FGDB_022SAE001@AddOn".AddT.Kick_out )
      wire#w3
      Coil( "022SAE001-SF2:X1" )
   END_RUNG
   RUNG wire#w1
      Contact( "022SAE001-SF5:22" )
   END_RUNG wire#w2
   RUNG wire#powerrail
      Contact( "FGDB_022SAE001@AddOn".AddT.Kick_in_two_side )
   END_RUNG wire#w3
   RUNG wire#powerrail
      Contact( "FGDB_001BR_010".TmrB."1_Run" )
   END_RUNG wire#w3
   // the same network as SCL:
   "022SAE001-SF2:X1" := ("Clock_1Hz" AND "022SAE001-SF6:14" AND ("022SAE001-SF5:14" OR "022SAE001-SF5:22") AND NOT "FGDB_022SAE001@AddOn".AddT.Kick_in_two_side AND NOT "FGDB_022SAE001@AddOn".AddT.Kick_in_one_side AND NOT "FGDB_022SAE001@AddOn".AddT.Kick_out) OR "FGDB_022SAE001@AddOn".AddT.Kick_in_two_side OR "FGDB_001BR_010".TmrB."1_Run";
END_REGION

REGION Network 23: 022SAE001 Confirm selection one side / Vorzeigen
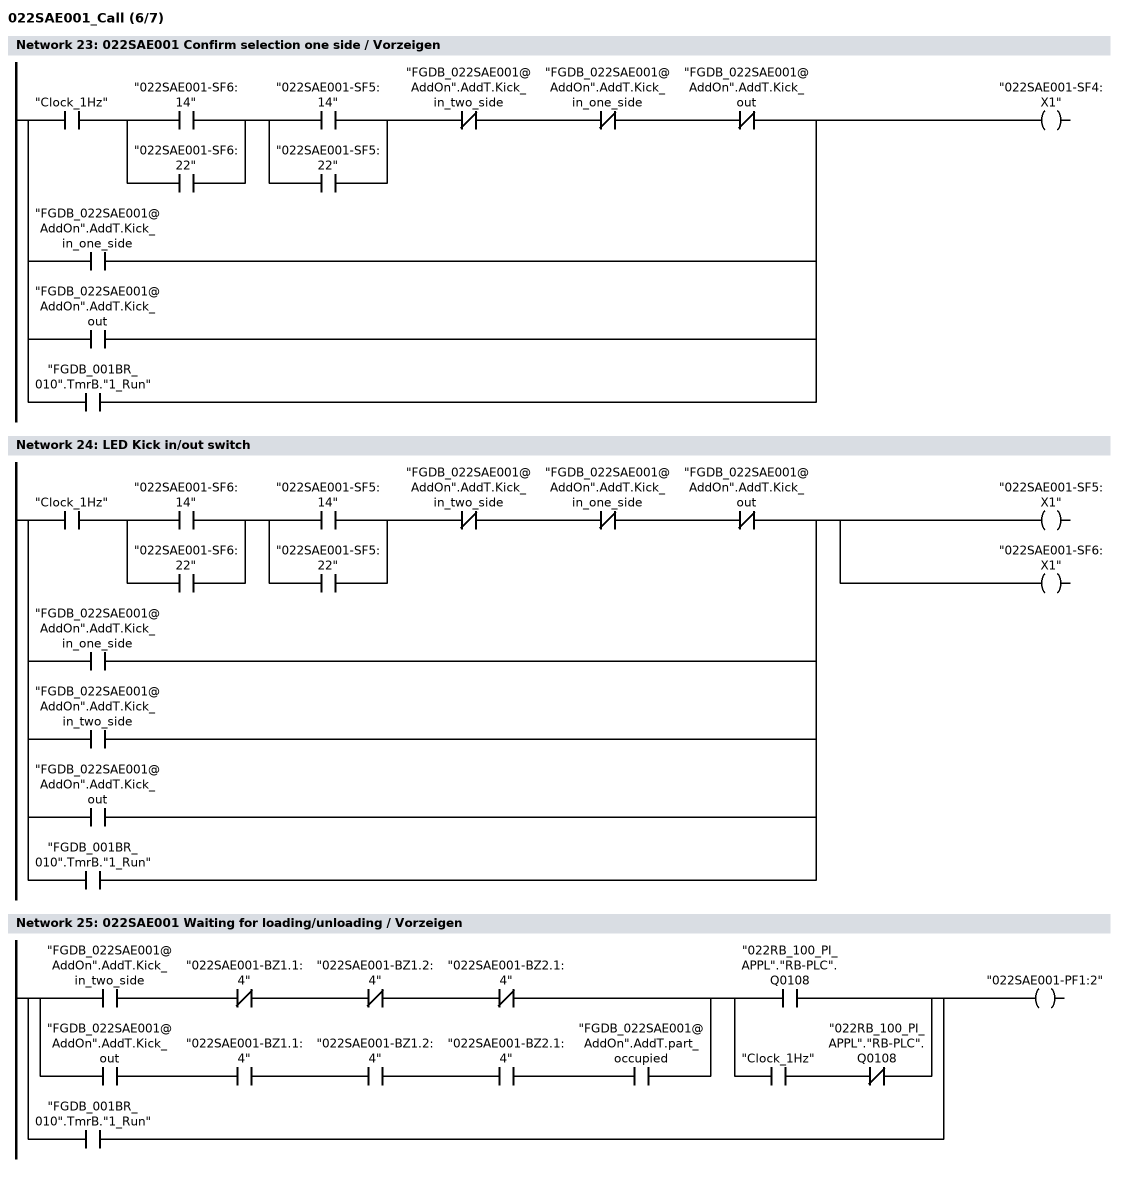
   RUNG wire#powerrail
      Contact( "Clock_1Hz" )
      wire#w1
      Contact( "022SAE001-SF6:14" )
      wire#w2
      Contact( "022SAE001-SF5:14" )
      wire#w3
      I_Contact( "FGDB_022SAE001@AddOn".AddT.Kick_in_two_side )
      I_Contact( "FGDB_022SAE001@AddOn".AddT.Kick_in_one_side )
      I_Contact( "FGDB_022SAE001@AddOn".AddT.Kick_out )
      wire#w4
      Coil( "022SAE001-SF4:X1" )
   END_RUNG
   RUNG wire#w1
      Contact( "022SAE001-SF6:22" )
   END_RUNG wire#w2
   RUNG wire#w2
      Contact( "022SAE001-SF5:22" )
   END_RUNG wire#w3
   RUNG wire#powerrail
      Contact( "FGDB_022SAE001@AddOn".AddT.Kick_in_one_side )
   END_RUNG wire#w4
   RUNG wire#powerrail
      Contact( "FGDB_022SAE001@AddOn".AddT.Kick_out )
   END_RUNG wire#w4
   RUNG wire#powerrail
      Contact( "FGDB_001BR_010".TmrB."1_Run" )
   END_RUNG wire#w4
   // the same network as SCL:
   "022SAE001-SF4:X1" := ("Clock_1Hz" AND ("022SAE001-SF6:14" OR "022SAE001-SF6:22") AND ("022SAE001-SF5:14" OR "022SAE001-SF5:22") AND NOT "FGDB_022SAE001@AddOn".AddT.Kick_in_two_side AND NOT "FGDB_022SAE001@AddOn".AddT.Kick_in_one_side AND NOT "FGDB_022SAE001@AddOn".AddT.Kick_out) OR "FGDB_022SAE001@AddOn".AddT.Kick_in_one_side OR "FGDB_022SAE001@AddOn".AddT.Kick_out OR "FGDB_001BR_010".TmrB."1_Run";
END_REGION

REGION Network 24: LED Kick in/out switch
   RUNG wire#powerrail
      Contact( "Clock_1Hz" )
      wire#w1
      Contact( "022SAE001-SF6:14" )
      wire#w2
      Contact( "022SAE001-SF5:14" )
      wire#w3
      I_Contact( "FGDB_022SAE001@AddOn".AddT.Kick_in_two_side )
      I_Contact( "FGDB_022SAE001@AddOn".AddT.Kick_in_one_side )
      I_Contact( "FGDB_022SAE001@AddOn".AddT.Kick_out )
      wire#w4
      Coil( "022SAE001-SF5:X1" )
   END_RUNG
   RUNG wire#w1
      Contact( "022SAE001-SF6:22" )
   END_RUNG wire#w2
   RUNG wire#w2
      Contact( "022SAE001-SF5:22" )
   END_RUNG wire#w3
   RUNG wire#powerrail
      Contact( "FGDB_022SAE001@AddOn".AddT.Kick_in_one_side )
   END_RUNG wire#w4
   RUNG wire#powerrail
      Contact( "FGDB_022SAE001@AddOn".AddT.Kick_in_two_side )
   END_RUNG wire#w4
   RUNG wire#powerrail
      Contact( "FGDB_022SAE001@AddOn".AddT.Kick_out )
   END_RUNG wire#w4
   RUNG wire#powerrail
      Contact( "FGDB_001BR_010".TmrB."1_Run" )
   END_RUNG wire#w4
   RUNG wire#w4
      Coil( "022SAE001-SF6:X1" )
   END_RUNG
   // the same network as SCL:
   "022SAE001-SF5:X1" := ("Clock_1Hz" AND ("022SAE001-SF6:14" OR "022SAE001-SF6:22") AND ("022SAE001-SF5:14" OR "022SAE001-SF5:22") AND NOT "FGDB_022SAE001@AddOn".AddT.Kick_in_two_side AND NOT "FGDB_022SAE001@AddOn".AddT.Kick_in_one_side AND NOT "FGDB_022SAE001@AddOn".AddT.Kick_out) OR "FGDB_022SAE001@AddOn".AddT.Kick_in_one_side OR "FGDB_022SAE001@AddOn".AddT.Kick_in_two_side OR "FGDB_022SAE001@AddOn".AddT.Kick_out OR "FGDB_001BR_010".TmrB."1_Run";
   "022SAE001-SF6:X1" := "022SAE001-SF5:X1";
END_REGION

REGION Network 25: 022SAE001 Waiting for loading/unloading / Vorzeigen
   RUNG wire#powerrail
      Contact( "FGDB_022SAE001@AddOn".AddT.Kick_in_two_side )
      I_Contact( "022SAE001-BZ1.1:4" )
      I_Contact( "022SAE001-BZ1.2:4" )
      I_Contact( "022SAE001-BZ2.1:4" )
      wire#w1
      Contact( "022RB_100_PI_APPL"."RB-PLC".Q0108 )
      wire#w2
      Coil( "022SAE001-PF1:2" )
   END_RUNG
   RUNG wire#powerrail
      Contact( "FGDB_022SAE001@AddOn".AddT.Kick_out )
      Contact( "022SAE001-BZ1.1:4" )
      Contact( "022SAE001-BZ1.2:4" )
      Contact( "022SAE001-BZ2.1:4" )
      Contact( "FGDB_022SAE001@AddOn".AddT.part_occupied )
   END_RUNG wire#w1
   RUNG wire#w1
      Contact( "Clock_1Hz" )
      I_Contact( "022RB_100_PI_APPL"."RB-PLC".Q0108 )
   END_RUNG wire#w2
   RUNG wire#powerrail
      Contact( "FGDB_001BR_010".TmrB."1_Run" )
   END_RUNG wire#w2
   // the same network as SCL:
   "022SAE001-PF1:2" := ((("FGDB_022SAE001@AddOn".AddT.Kick_in_two_side AND NOT "022SAE001-BZ1.1:4" AND NOT "022SAE001-BZ1.2:4" AND NOT "022SAE001-BZ2.1:4") OR ("FGDB_022SAE001@AddOn".AddT.Kick_out AND "022SAE001-BZ1.1:4" AND "022SAE001-BZ1.2:4" AND "022SAE001-BZ2.1:4" AND "FGDB_022SAE001@AddOn".AddT.part_occupied)) AND ("022RB_100_PI_APPL"."RB-PLC".Q0108 OR ("Clock_1Hz" AND NOT "022RB_100_PI_APPL"."RB-PLC".Q0108))) OR "FGDB_001BR_010".TmrB."1_Run";
END_REGION

REGION Network 26: 022SAE001 Part in position and kick out select / Vorzeigen
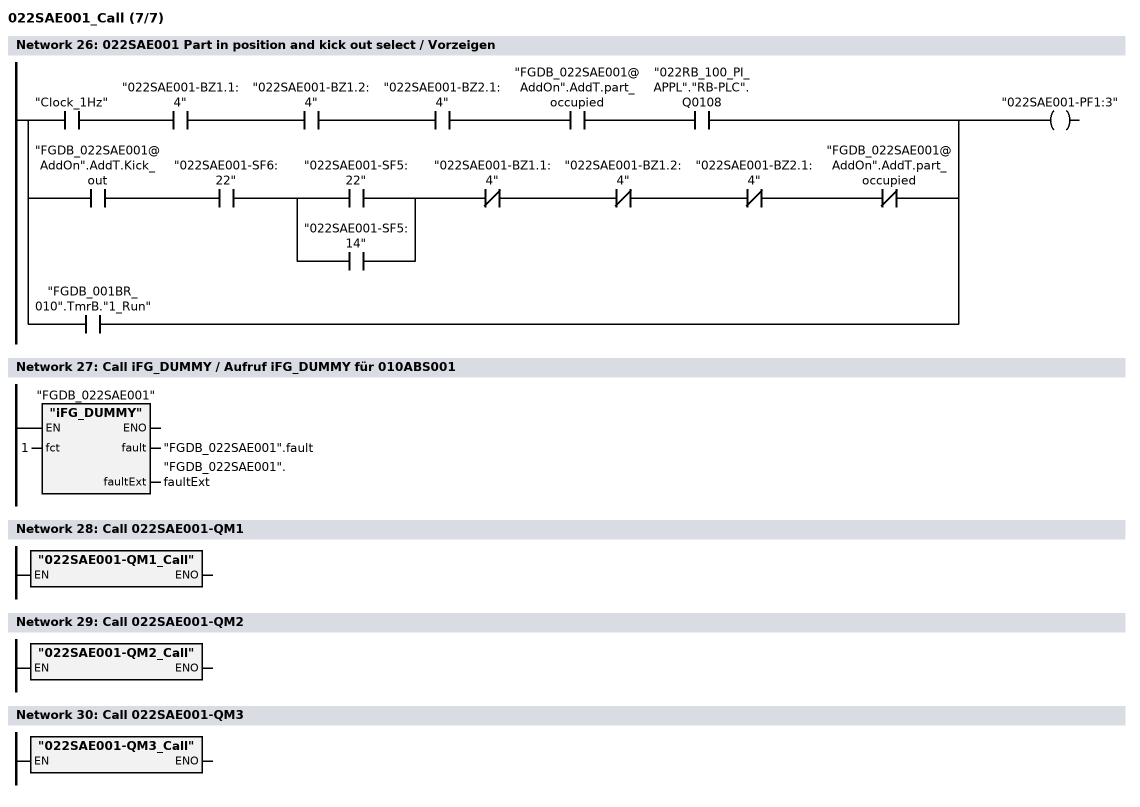
   RUNG wire#powerrail
      Contact( "Clock_1Hz" )
      Contact( "022SAE001-BZ1.1:4" )
      Contact( "022SAE001-BZ1.2:4" )
      Contact( "022SAE001-BZ2.1:4" )
      Contact( "FGDB_022SAE001@AddOn".AddT.part_occupied )
      Contact( "022RB_100_PI_APPL"."RB-PLC".Q0108 )
      wire#w1
      Coil( "022SAE001-PF1:3" )
   END_RUNG
   RUNG wire#powerrail
      Contact( "FGDB_022SAE001@AddOn".AddT.Kick_out )
      Contact( "022SAE001-SF6:22" )
      wire#w2
      Contact( "022SAE001-SF5:22" )
      wire#w3
      I_Contact( "022SAE001-BZ1.1:4" )
      I_Contact( "022SAE001-BZ1.2:4" )
      I_Contact( "022SAE001-BZ2.1:4" )
      I_Contact( "FGDB_022SAE001@AddOn".AddT.part_occupied )
   END_RUNG wire#w1
   RUNG wire#w2
      Contact( "022SAE001-SF5:14" )
   END_RUNG wire#w3
   RUNG wire#powerrail
      Contact( "FGDB_001BR_010".TmrB."1_Run" )
   END_RUNG wire#w1
   // the same network as SCL:
   "022SAE001-PF1:3" := ("Clock_1Hz" AND "022SAE001-BZ1.1:4" AND "022SAE001-BZ1.2:4" AND "022SAE001-BZ2.1:4" AND "FGDB_022SAE001@AddOn".AddT.part_occupied AND "022RB_100_PI_APPL"."RB-PLC".Q0108) OR ("FGDB_022SAE001@AddOn".AddT.Kick_out AND "022SAE001-SF6:22" AND ("022SAE001-SF5:22" OR "022SAE001-SF5:14") AND NOT "022SAE001-BZ1.1:4" AND NOT "022SAE001-BZ1.2:4" AND NOT "022SAE001-BZ2.1:4" AND NOT "FGDB_022SAE001@AddOn".AddT.part_occupied) OR "FGDB_001BR_010".TmrB."1_Run";
END_REGION

REGION Network 27: Call iFG_DUMMY / Aufruf iFG_DUMMY für 010ABS001
   RUNG wire#powerrail
      "FGDB_022SAE001"(fct := 1, fault => "FGDB_022SAE001".fault, faultExt => "FGDB_022SAE001".faultExt)
   END_RUNG
   // the same network as SCL:
   "FGDB_022SAE001"(fct := 1, fault => "FGDB_022SAE001".fault, faultExt => "FGDB_022SAE001".faultExt);   // "iFG_DUMMY"
END_REGION

REGION Network 28: Call 022SAE001-QM1
   RUNG wire#powerrail
      "022SAE001-QM1_Call"()
   END_RUNG
   // the same network as SCL:
   "022SAE001-QM1_Call"();
END_REGION

REGION Network 29: Call 022SAE001-QM2
   RUNG wire#powerrail
      "022SAE001-QM2_Call"()
   END_RUNG
   // the same network as SCL:
   "022SAE001-QM2_Call"();
END_REGION

REGION Network 30: Call 022SAE001-QM3
   RUNG wire#powerrail
      "022SAE001-QM3_Call"()
   END_RUNG
   // the same network as SCL:
   "022SAE001-QM3_Call"();
END_REGION
END_FUNCTION
